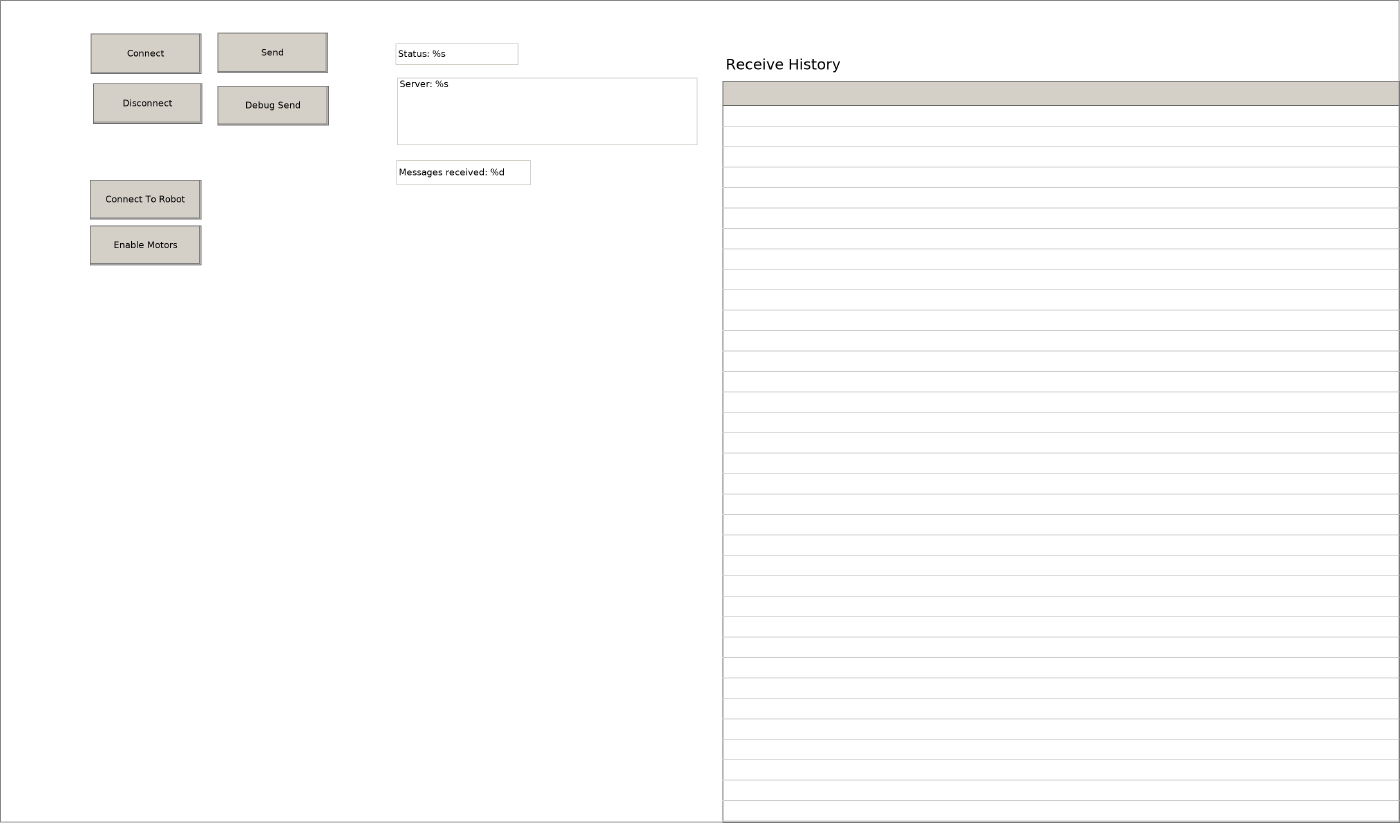
VISUALIZATION VisualizationControlPanel  // 1713x1007
    Button (114,102 133x49), "Disconnect"
        tap MAIN.buttonDisconnectPressed
    Button (266,40 135x49), "Send"
        tap MAIN.buttonSendPressed
    Button (111,41 135x49), "Connect"
        tap MAIN.buttonConnectPressed
    Textfield (486,95 367x82), "Server: %s", text variable: MAIN.messageFromServer
    Textfield (485,196 164x30), "Messages received: %d", text variable: MAIN.totalMessagesFromServerCount
    Table (884,99 829x908), data array: MAIN.messageHistoryArray
        p3854506369: MAIN.messageHistoryArray[INDEX].systemTimeString
        p1892666644: MAIN.messageHistoryArray[INDEX].message
        p511219082: Message
    Label (885,64 182x30), "Receive History"
    Button (110,220 136x48), "Connect To Robot"
        tap MAIN.buttonConnectToRobotPressed
    Button (266,105 136x48), "Debug Send"
        tap MAIN.buttonDebugSendPressed
    Button (110,276 136x48), "Enable Motors"
        tap MAIN.buttonEnableMotorsPressed
    Textfield (484,53 150x26), "Status: %s", text variable: MAIN.connectionMessage
END_VISUALIZATION

(* stored: Version 1.1.0.1, ProductVersion 3.1.4024.12
   Visu VisualizationControlPanel: Id {65fbdb0c-c9af-43b6-9432-86e4c4c3ac9b} *)
